FUNCTION BYTE_TO_ARR08B
  (* Standard: 61499-1 *)
  (* Version 1.0, 2024-02-22, franz *)
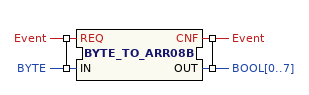
  EVENT_INPUT
    REQ WITH IN; (* Normal Execution Request *)
  END_EVENT
  EVENT_OUTPUT
    CNF WITH OUT; (* Execution Confirmation *)
  END_EVENT
  VAR_INPUT
    IN : BYTE; (* BYTE Input *)
  END_VAR
  VAR_OUTPUT
    OUT : ARRAY [0..7] OF BOOL; (* ARR08B Output *)
  END_VAR
  BODY IN ST:
FUNCTION BYTE_TO_ARR08B

VAR_INPUT
	IN : BYTE;    // BYTE Input
END_VAR

VAR_OUTPUT
	OUT : ARRAY[0..7] OF BOOL;    // ARR08B Output
END_VAR

(* this Function extracts the 8 Bits from a byte *)
OUT[0] := IN.0;
OUT[1] := IN.1;
OUT[2] := IN.2;
OUT[3] := IN.3;
OUT[4] := IN.4;
OUT[5] := IN.5;
OUT[6] := IN.6;
OUT[7] := IN.7;

END_FUNCTION
  END_BODY
END_FUNCTION
